// TIA Portal V18 export
// export: Created 2026-06-13T06:09:46.0384425Z, ExportSetting WithDefaults, DisplayName Totally Integrated Automation Portal, DisplayVersion V18, DisplayName TIA Portal Openness, DisplayVersion V18, DisplayName TIA Portal Version Control Interface, DisplayVersion V18, DisplayName STEP 7 Professional, DisplayVersion V18, DisplayName STEP 7 Safety, DisplayVersion V18, DisplayName WinCC Professional, DisplayVersion V18
ORGANIZATION_BLOCK "OB30_PID_PLC1_Bon2"   // OB30, LAD, CyclicInterrupt
{ S7_Optimized_Access := 'TRUE' }
VERSION : 0.1
// stored: AutoNumber true, IsIECCheckEnabled false, SetENOAutomatically false
   VAR_INPUT
      Initial_Call : Bool;   // Initial call of this OB
      Event_Count : Int;   // Events discarded
   END_VAR
BEGIN

REGION Network 1: Initialize PID Bon 2 Kp parameter
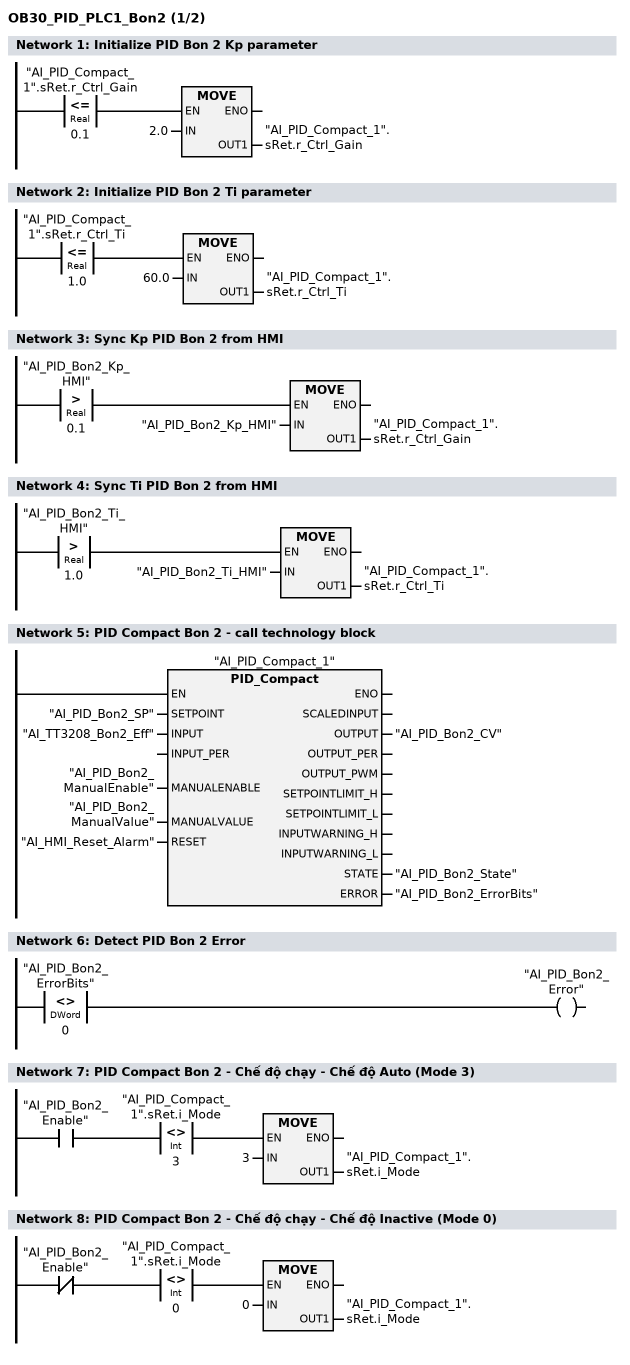
   RUNG wire#powerrail
      { S7_Templates := "SrcType := Real" } LE_Contact(in1 := "AI_PID_Compact_1".sRet.r_Ctrl_Gain, in2 := 0.1)
      { S7_GenerateENO := "TRUE" } Move(in := 2.0, out1 => "AI_PID_Compact_1".sRet.r_Ctrl_Gain)
   END_RUNG
   // the same network as SCL:
   IF "AI_PID_Compact_1".sRet.r_Ctrl_Gain <= 0.1 THEN "AI_PID_Compact_1".sRet.r_Ctrl_Gain := 2.0; END_IF;
END_REGION

REGION Network 2: Initialize PID Bon 2 Ti parameter
   RUNG wire#powerrail
      { S7_Templates := "SrcType := Real" } LE_Contact(in1 := "AI_PID_Compact_1".sRet.r_Ctrl_Ti, in2 := 1.0)
      { S7_GenerateENO := "TRUE" } Move(in := 60.0, out1 => "AI_PID_Compact_1".sRet.r_Ctrl_Ti)
   END_RUNG
   // the same network as SCL:
   IF "AI_PID_Compact_1".sRet.r_Ctrl_Ti <= 1.0 THEN "AI_PID_Compact_1".sRet.r_Ctrl_Ti := 60.0; END_IF;
END_REGION

REGION Network 3: Sync Kp PID Bon 2 from HMI
   RUNG wire#powerrail
      { S7_Templates := "SrcType := Real" } GT_Contact(in1 := "AI_PID_Bon2_Kp_HMI", in2 := 0.1)
      { S7_GenerateENO := "TRUE" } Move(in := "AI_PID_Bon2_Kp_HMI", out1 => "AI_PID_Compact_1".sRet.r_Ctrl_Gain)
   END_RUNG
   // the same network as SCL:
   IF "AI_PID_Bon2_Kp_HMI" > 0.1 THEN "AI_PID_Compact_1".sRet.r_Ctrl_Gain := "AI_PID_Bon2_Kp_HMI"; END_IF;
END_REGION

REGION Network 4: Sync Ti PID Bon 2 from HMI
   RUNG wire#powerrail
      { S7_Templates := "SrcType := Real" } GT_Contact(in1 := "AI_PID_Bon2_Ti_HMI", in2 := 1.0)
      { S7_GenerateENO := "TRUE" } Move(in := "AI_PID_Bon2_Ti_HMI", out1 => "AI_PID_Compact_1".sRet.r_Ctrl_Ti)
   END_RUNG
   // the same network as SCL:
   IF "AI_PID_Bon2_Ti_HMI" > 1.0 THEN "AI_PID_Compact_1".sRet.r_Ctrl_Ti := "AI_PID_Bon2_Ti_HMI"; END_IF;
END_REGION

REGION Network 5: PID Compact Bon 2 - call technology block
   RUNG wire#powerrail
      "AI_PID_Compact_1".PID_Compact(Setpoint := "AI_PID_Bon2_SP", Input := "AI_TT3208_Bon2_Eff", Input_PER :=, ManualEnable := "AI_PID_Bon2_ManualEnable", ManualValue := "AI_PID_Bon2_ManualValue", Reset := "AI_HMI_Reset_Alarm", ScaledInput =>, Output => "AI_PID_Bon2_CV", Output_PER =>, Output_PWM =>, SetpointLimit_H =>, SetpointLimit_L =>, InputWarning_H =>, InputWarning_L =>, State => "AI_PID_Bon2_State", Error => "AI_PID_Bon2_ErrorBits")
   END_RUNG
   // the same network as SCL:
   "AI_PID_Compact_1"(Setpoint := "AI_PID_Bon2_SP",   // PID_Compact
                      Input := "AI_TT3208_Bon2_Eff",
                      ManualEnable := "AI_PID_Bon2_ManualEnable",
                      ManualValue := "AI_PID_Bon2_ManualValue",
                      Reset := "AI_HMI_Reset_Alarm",
                      Output => "AI_PID_Bon2_CV",
                      State => "AI_PID_Bon2_State",
                      Error => "AI_PID_Bon2_ErrorBits");
END_REGION

REGION Network 6: Detect PID Bon 2 Error
   RUNG wire#powerrail
      { S7_Templates := "SrcType := DWord" } NE_Contact(in1 := "AI_PID_Bon2_ErrorBits", in2 := 0)
      Coil( "AI_PID_Bon2_Error" )
   END_RUNG
   // the same network as SCL:
   "AI_PID_Bon2_Error" := "AI_PID_Bon2_ErrorBits" <> 0;
END_REGION

REGION Network 7: PID Compact Bon 2 - Chế độ chạy - Chế độ Auto (Mode 3)
   RUNG wire#powerrail
      Contact( "AI_PID_Bon2_Enable" )
      { S7_Templates := "SrcType := Int" } NE_Contact(in1 := "AI_PID_Compact_1".sRet.i_Mode, in2 := 3)
      { S7_GenerateENO := "TRUE" } Move(in := 3, out1 => "AI_PID_Compact_1".sRet.i_Mode)
   END_RUNG
   // the same network as SCL:
   IF "AI_PID_Bon2_Enable" AND ("AI_PID_Compact_1".sRet.i_Mode <> 3) THEN
       "AI_PID_Compact_1".sRet.i_Mode := 3;
   END_IF;
END_REGION

REGION Network 8: PID Compact Bon 2 - Chế độ chạy - Chế độ Inactive (Mode 0)
   RUNG wire#powerrail
      I_Contact( "AI_PID_Bon2_Enable" )
      { S7_Templates := "SrcType := Int" } NE_Contact(in1 := "AI_PID_Compact_1".sRet.i_Mode, in2 := 0)
      { S7_GenerateENO := "TRUE" } Move(in := 0, out1 => "AI_PID_Compact_1".sRet.i_Mode)
   END_RUNG
   // the same network as SCL:
   IF NOT "AI_PID_Bon2_Enable" AND ("AI_PID_Compact_1".sRet.i_Mode <> 0) THEN
       "AI_PID_Compact_1".sRet.i_Mode := 0;
   END_IF;
END_REGION

REGION Network 9: Move PID Bon 2 CV to Steam Valve
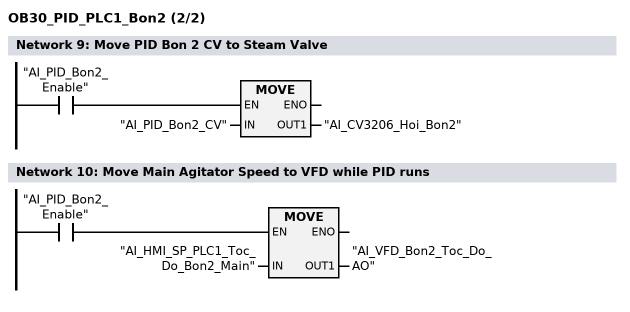
   RUNG wire#powerrail
      Contact( "AI_PID_Bon2_Enable" )
      { S7_GenerateENO := "TRUE" } Move(in := "AI_PID_Bon2_CV", out1 => "AI_CV3206_Hoi_Bon2")
   END_RUNG
   // the same network as SCL:
   IF "AI_PID_Bon2_Enable" THEN "AI_CV3206_Hoi_Bon2" := "AI_PID_Bon2_CV"; END_IF;
END_REGION

REGION Network 10: Move Main Agitator Speed to VFD while PID runs
   RUNG wire#powerrail
      Contact( "AI_PID_Bon2_Enable" )
      { S7_GenerateENO := "TRUE" } Move(in := "AI_HMI_SP_PLC1_Toc_Do_Bon2_Main", out1 => "AI_VFD_Bon2_Toc_Do_AO")
   END_RUNG
   // the same network as SCL:
   IF "AI_PID_Bon2_Enable" THEN "AI_VFD_Bon2_Toc_Do_AO" := "AI_HMI_SP_PLC1_Toc_Do_Bon2_Main"; END_IF;
END_REGION
END_ORGANIZATION_BLOCK
